FUNCTION Disable_Axis : INT

VAR_INPUT

END_VAR

VAR_IN_OUT
	Axis: Motion_Axis;
END_VAR

VAR

END_VAR

Axis.IN_Enable_Control:= 0;
Axis.OL_IN_Analog:= 0;
Axis.CL_IN_Vel:= 0;
Axis.OL_IN_Slave_Enable:= 0;
Axis.OL_IN_Slave_Command:= 0;
Axis.CL_IN_Slave_Enable:= 0;
Axis.CL_IN_Slave_Command:= 0;
Axis.IN_Func_1:= 0;	//Should these be here?
Axis.IN_Func_2:= 0;	//Should these be here?	
Axis.IN_Func_3:= 0;	//Should these be here?	
Axis.IN_Func_4:= 0;	//Should these be here?	
Axis.OL_IN_Bump_Duration:= T#0MS; 
Axis.OL_IN_Bump_Trigger:= 0;
Axis.CL_RUN_Position_Reached:=0;

END_FUNCTION

(* stored: Version 1.1.0.1, ProductVersion 3.1.4024.0
   POU Disable_Axis: Id {0eef292d-6f9c-47bf-b4ee-8643e75fdfd3}, SpecialFunc None *)
